TYPE IRecipe :
STRUCT
	bCreate:BOOL;
	bSave:BOOL;
	bLoad:BOOL;

     
END_STRUCT
END_TYPE

(* stored: Version 1.1.0.1, ProductVersion 3.1.4024.9
   DUT IRecipe: Id {4665c4c1-ee89-4ce8-9429-07c93214e90f} *)
